// TIA Portal V18 export
FUNCTION_BLOCK "TD_Control"   // FB19, LAD
TITLE = TD_Control
{ S7_Optimized_Access := 'TRUE' }
// Written BY Kristopher Gimenez Feb1,2023
// This block is used to control the TD control mode, pump outputs and HSLT/LSHT shifting
// stored: AutoNumber false, MemoryReserve 100, SetENOAutomatically false
   VAR
      AllowShift : Bool;   // Allow speed change
      TD_Mode : Int;   // TD Mode, 0=Drill, 1=DrillRev, 2=MU-S, 3=MU-T, 4= BO, 5 OSC, 6 Bypass
      HSLTShift_TP { S7_SetPoint := 'True'} : TP_TIME;
      LSHTShift_TP { S7_SetPoint := 'True'} : TP_TIME;
      MUSpinComplete : Bool;   // Set once MU spin torq above setpoint
      TDP1FwdSetmA : Real;
      TDP2FwdSetmA : Real;
      TDP1RevSetmA : Real;
      TDP2RevSetmA : Real;
      TorqSetmA : Real;
      TDP1FwdEn : Bool;
      TDP2FwdEn : Bool;
      TDP1RevEn : Bool;
      TDP2RevEn : Bool;
      TorqEn : Bool;
      BypassDelay_TON { S7_SetPoint := 'True'} : TON_TIME;
      BypassRunning_TOF { S7_SetPoint := 'True'} : TOF_TIME;
      HSLT_Sol_Last { S7_SetPoint := 'True'} : Bool;
      LSHT_Sol_Last : Bool;
      AllowRev : Bool;   // Latch that will allow Drill rev if rotary has stopped
      SpeedLimiting : Bool;
      SpeedLimitmAOut : Real;
      SpeedLimitingTrig : Bool;   // Positive Trigger Last cycle value
      MUTorqStart : Bool;
      BOStart : Bool;
      OscStart : Bool;
      MUTorqStart_Trig : Bool;
      BOStart_Trig : Bool;
      OscStart_Trig : Bool;
      SpeedLimit_SlewDec { S7_SetPoint := 'True'} : "SlewDec";
      SpeedLimit_SlewInc { S7_SetPoint := 'True'} : "SlewInc";
      HiTempShutDown_TON { S7_SetPoint := 'True'} : TON_TIME;
   END_VAR
   VAR_TEMP
      FlowmAOutTemp : Real;
      TorqmAOutTemp : Real;
      TorqPSITemp : Real;
      TorquePSI : Real;
      tempReal : Real;
   END_VAR
   VAR CONSTANT
      Disabled : Int := 0;   // TD Mode State Machine
      Drill : Int := 1;   // TD Mode State Machine
      DrillReverse : Int := 2;   // TD Mode State Machine
      MUSpin : Int := 3;   // TD Mode State Machine
      MUTorq : Int := 4;   // TD Mode State Machine
      BO : Int := 5;   // TD Mode State Machine
      Oscillate : Int := 6;   // TD Mode State Machine
      Bypass : Int := 7;   // TD Mode State Machine
   END_VAR
   VAR_TEMP   // added for the SCL form of the ladder/FBD networks
      _w1 : Bool;
      _w2 : Bool;
      _w3 : Bool;
      _w4 : Bool;
   END_VAR
BEGIN

REGION Network 1: Control Mode
   // Determine Control Mode based on Console Inputs and interlocks.
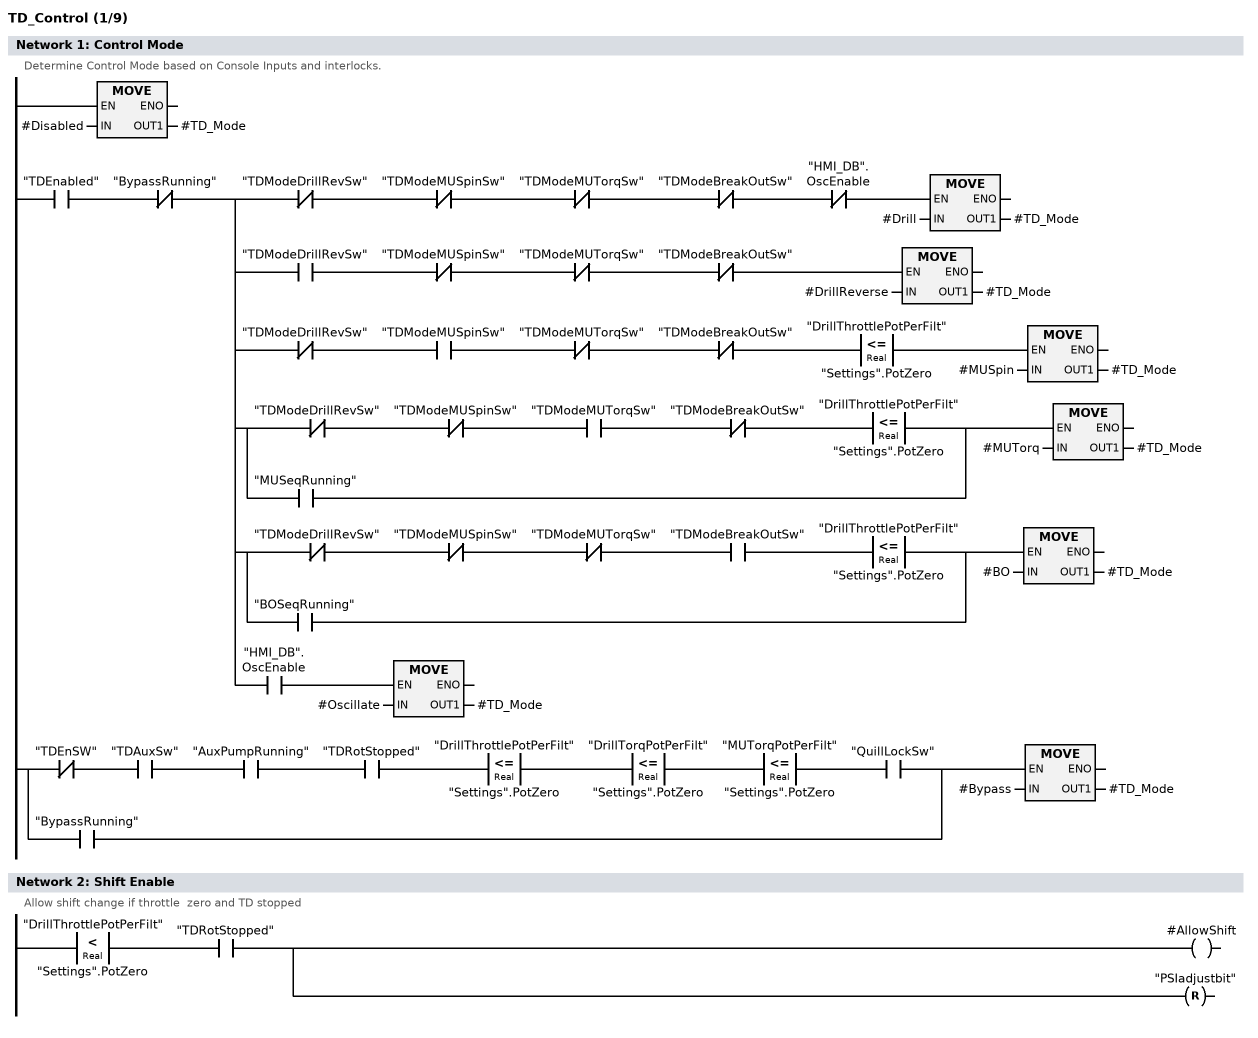
   RUNG wire#powerrail
      Move(in := #Disabled, out1 => #TD_Mode)
   END_RUNG
   RUNG wire#powerrail
      Contact( "TDEnabled" )
      I_Contact( "BypassRunning" )
      wire#w1
      I_Contact( "TDModeDrillRevSw" )
      I_Contact( "TDModeMUSpinSw" )
      I_Contact( "TDModeMUTorqSw" )
      I_Contact( "TDModeBreakOutSw" )
      I_Contact( "HMI_DB".OscEnable )
      Move(in := #Drill, out1 => #TD_Mode)
   END_RUNG
   RUNG wire#w1
      Contact( "TDModeDrillRevSw" )
      I_Contact( "TDModeMUSpinSw" )
      I_Contact( "TDModeMUTorqSw" )
      I_Contact( "TDModeBreakOutSw" )
      Move(in := #DrillReverse, out1 => #TD_Mode)
   END_RUNG
   RUNG wire#w1
      I_Contact( "TDModeDrillRevSw" )
      Contact( "TDModeMUSpinSw" )
      I_Contact( "TDModeMUTorqSw" )
      I_Contact( "TDModeBreakOutSw" )
      { S7_Templates := "SrcType := Real" } LE_Contact(in1 := "DrillThrottlePotPerFilt", in2 := "Settings".PotZero)
      Move(in := #MUSpin, out1 => #TD_Mode)
   END_RUNG
   RUNG wire#w1
      I_Contact( "TDModeDrillRevSw" )
      I_Contact( "TDModeMUSpinSw" )
      Contact( "TDModeMUTorqSw" )
      I_Contact( "TDModeBreakOutSw" )
      { S7_Templates := "SrcType := Real" } LE_Contact(in1 := "DrillThrottlePotPerFilt", in2 := "Settings".PotZero)
      wire#w2
      Move(in := #MUTorq, out1 => #TD_Mode)
   END_RUNG
   RUNG wire#w1
      Contact( "MUSeqRunning" )
   END_RUNG wire#w2
   RUNG wire#w1
      I_Contact( "TDModeDrillRevSw" )
      I_Contact( "TDModeMUSpinSw" )
      I_Contact( "TDModeMUTorqSw" )
      Contact( "TDModeBreakOutSw" )
      { S7_Templates := "SrcType := Real" } LE_Contact(in1 := "DrillThrottlePotPerFilt", in2 := "Settings".PotZero)
      wire#w3
      Move(in := #BO, out1 => #TD_Mode)
   END_RUNG
   RUNG wire#w1
      Contact( "BOSeqRunning" )
   END_RUNG wire#w3
   RUNG wire#w1
      Contact( "HMI_DB".OscEnable )
      Move(in := #Oscillate, out1 => #TD_Mode)
   END_RUNG
   RUNG wire#powerrail
      I_Contact( "TDEnSW" )
      Contact( "TDAuxSw" )
      Contact( "AuxPumpRunning" )
      Contact( "TDRotStopped" )
      { S7_Templates := "SrcType := Real" } LE_Contact(in1 := "DrillThrottlePotPerFilt", in2 := "Settings".PotZero)
      { S7_Templates := "SrcType := Real" } LE_Contact(in1 := "DrillTorqPotPerFilt", in2 := "Settings".PotZero)
      { S7_Templates := "SrcType := Real" } LE_Contact(in1 := "MUTorqPotPerFilt", in2 := "Settings".PotZero)
      Contact( "QuillLockSw" )
      wire#w4
      Move(in := #Bypass, out1 => #TD_Mode)
   END_RUNG
   RUNG wire#powerrail
      Contact( "BypassRunning" )
   END_RUNG wire#w4
   // the same network as SCL:
   #TD_Mode := #Disabled;
   #_w1 := "TDEnabled" AND NOT "BypassRunning";
   IF #_w1 AND NOT "TDModeDrillRevSw" AND NOT "TDModeMUSpinSw" AND NOT "TDModeMUTorqSw" AND NOT "TDModeBreakOutSw" AND NOT "HMI_DB".OscEnable THEN
       #TD_Mode := #Drill;
   END_IF;
   IF #_w1 AND "TDModeDrillRevSw" AND NOT "TDModeMUSpinSw" AND NOT "TDModeMUTorqSw" AND NOT "TDModeBreakOutSw" THEN
       #TD_Mode := #DrillReverse;
   END_IF;
   IF #_w1 AND NOT "TDModeDrillRevSw" AND "TDModeMUSpinSw" AND NOT "TDModeMUTorqSw" AND NOT "TDModeBreakOutSw" AND ("DrillThrottlePotPerFilt" <= "Settings".PotZero) THEN
       #TD_Mode := #MUSpin;
   END_IF;
   IF #_w1 AND ((NOT "TDModeDrillRevSw" AND NOT "TDModeMUSpinSw" AND "TDModeMUTorqSw" AND NOT "TDModeBreakOutSw" AND ("DrillThrottlePotPerFilt" <= "Settings".PotZero)) OR "MUSeqRunning") THEN
       #TD_Mode := #MUTorq;
   END_IF;
   IF #_w1 AND ((NOT "TDModeDrillRevSw" AND NOT "TDModeMUSpinSw" AND NOT "TDModeMUTorqSw" AND "TDModeBreakOutSw" AND ("DrillThrottlePotPerFilt" <= "Settings".PotZero)) OR "BOSeqRunning") THEN
       #TD_Mode := #BO;
   END_IF;
   IF #_w1 AND "HMI_DB".OscEnable THEN #TD_Mode := #Oscillate; END_IF;
   IF (NOT "TDEnSW" AND "TDAuxSw" AND "AuxPumpRunning" AND "TDRotStopped" AND ("DrillThrottlePotPerFilt" <= "Settings".PotZero) AND ("DrillTorqPotPerFilt" <= "Settings".PotZero) AND ("MUTorqPotPerFilt" <= "Settings".PotZero) AND "QuillLockSw") OR "BypassRunning" THEN
       #TD_Mode := #Bypass;
   END_IF;
END_REGION

REGION Network 2: Shift Enable
   // Allow shift change if throttle  zero and TD stopped
   RUNG wire#powerrail
      { S7_Templates := "SrcType := Real" } LT_Contact(in1 := "DrillThrottlePotPerFilt", in2 := "Settings".PotZero)
      Contact( "TDRotStopped" )
      wire#w1
      Coil( #AllowShift )
   END_RUNG
   RUNG wire#w1
      R_Coil( "PSIadjustbit" )
   END_RUNG
   // the same network as SCL:
   #AllowShift := ("DrillThrottlePotPerFilt" < "Settings".PotZero) AND "TDRotStopped";
   IF #AllowShift THEN "PSIadjustbit" := FALSE; END_IF;
END_REGION

REGION Network 3: HSLT/LSHT
   // Allow Shifting.  
   // Bypass in HSLT.  
   // MU modes, BO and Osc in LSHT. 
   // Drill modes follow console input
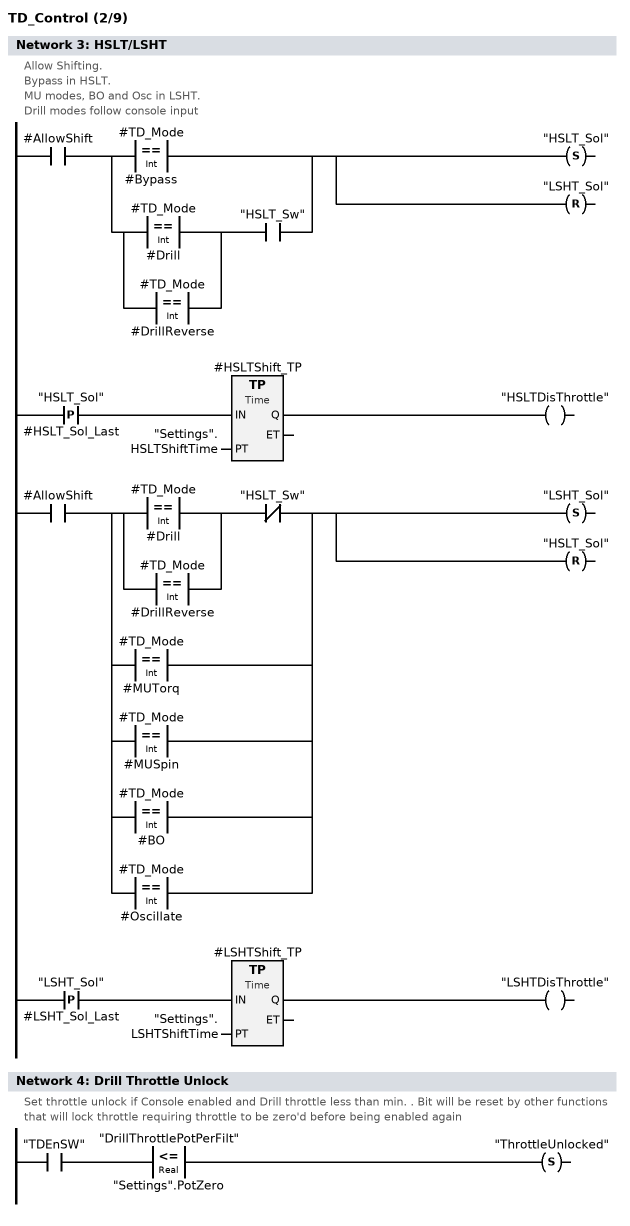
   RUNG wire#powerrail
      Contact( #AllowShift )
      wire#w1
      { S7_Templates := "SrcType := Int" } EQ_Contact(in1 := #TD_Mode, in2 := #Bypass)
      wire#w2
      S_Coil( "HSLT_Sol" )
   END_RUNG
   RUNG wire#w1
      { S7_Templates := "SrcType := Int" } EQ_Contact(in1 := #TD_Mode, in2 := #Drill)
      wire#w3
      Contact( "HSLT_Sw" )
   END_RUNG wire#w2
   RUNG wire#w1
      { S7_Templates := "SrcType := Int" } EQ_Contact(in1 := #TD_Mode, in2 := #DrillReverse)
   END_RUNG wire#w3
   RUNG wire#w2
      R_Coil( "LSHT_Sol" )
   END_RUNG
   RUNG wire#powerrail
      P_Contact(operand := "HSLT_Sol", bit := #HSLT_Sol_Last)
      { S7_Templates := "time_type := Time" } #HSLTShift_TP.TP(pt := "Settings".HSLTShiftTime, et =>)
      Coil( "HSLTDisThrottle" )
   END_RUNG
   RUNG wire#powerrail
      Contact( #AllowShift )
      wire#w4
      { S7_Templates := "SrcType := Int" } EQ_Contact(in1 := #TD_Mode, in2 := #Drill)
      wire#w5
      I_Contact( "HSLT_Sw" )
      wire#w6
      S_Coil( "LSHT_Sol" )
   END_RUNG
   RUNG wire#w4
      { S7_Templates := "SrcType := Int" } EQ_Contact(in1 := #TD_Mode, in2 := #DrillReverse)
   END_RUNG wire#w5
   RUNG wire#w4
      { S7_Templates := "SrcType := Int" } EQ_Contact(in1 := #TD_Mode, in2 := #MUTorq)
   END_RUNG wire#w6
   RUNG wire#w4
      { S7_Templates := "SrcType := Int" } EQ_Contact(in1 := #TD_Mode, in2 := #MUSpin)
   END_RUNG wire#w6
   RUNG wire#w4
      { S7_Templates := "SrcType := Int" } EQ_Contact(in1 := #TD_Mode, in2 := #BO)
   END_RUNG wire#w6
   RUNG wire#w4
      { S7_Templates := "SrcType := Int" } EQ_Contact(in1 := #TD_Mode, in2 := #Oscillate)
   END_RUNG wire#w6
   RUNG wire#w6
      R_Coil( "HSLT_Sol" )
   END_RUNG
   RUNG wire#powerrail
      P_Contact(operand := "LSHT_Sol", bit := #LSHT_Sol_Last)
      { S7_Templates := "time_type := Time" } #LSHTShift_TP.TP(pt := "Settings".LSHTShiftTime, et =>)
      Coil( "LSHTDisThrottle" )
   END_RUNG
   // the same network as SCL:
   IF #AllowShift AND ((#TD_Mode = #Bypass) OR (((#TD_Mode = #Drill) OR (#TD_Mode = #DrillReverse)) AND "HSLT_Sw")) THEN
       "HSLT_Sol" := TRUE;
       "LSHT_Sol" := FALSE;
   END_IF;
   #_w1 := "HSLT_Sol" AND NOT #HSLT_Sol_Last;   // rising edge of "HSLT_Sol"
   #HSLT_Sol_Last := "HSLT_Sol";
   #HSLTShift_TP(IN := #_w1, PT := "Settings".HSLTShiftTime);   // TP
   "HSLTDisThrottle" := #HSLTShift_TP.Q;
   IF #AllowShift AND ((((#TD_Mode = #Drill) OR (#TD_Mode = #DrillReverse)) AND NOT "HSLT_Sw") OR (#TD_Mode = #MUTorq) OR (#TD_Mode = #MUSpin) OR (#TD_Mode = #BO) OR (#TD_Mode = #Oscillate)) THEN
       "LSHT_Sol" := TRUE;
       "HSLT_Sol" := FALSE;
   END_IF;
   #_w2 := "LSHT_Sol" AND NOT #LSHT_Sol_Last;   // rising edge of "LSHT_Sol"
   #LSHT_Sol_Last := "LSHT_Sol";
   #LSHTShift_TP(IN := #_w2, PT := "Settings".LSHTShiftTime);   // TP
   "LSHTDisThrottle" := #LSHTShift_TP.Q;
END_REGION

REGION Network 4: Drill Throttle Unlock
   // Set throttle unlock if Console enabled and Drill throttle less than min. . Bit will be reset by other functions that will lock throttle requiring throttle to be zero'd before being enabled again
   RUNG wire#powerrail
      Contact( "TDEnSW" )
      { S7_Templates := "SrcType := Real" } LE_Contact(in1 := "DrillThrottlePotPerFilt", in2 := "Settings".PotZero)
      S_Coil( "ThrottleUnlocked" )
   END_RUNG
   // the same network as SCL:
   IF "TDEnSW" AND ("DrillThrottlePotPerFilt" <= "Settings".PotZero) THEN "ThrottleUnlocked" := TRUE; END_IF;
END_REGION

REGION Network 5: Drill Throttle Disable
   // Disable throttle if Bypass, Throttle disabled due to shift, or Flush fault or if throttle not unlocked
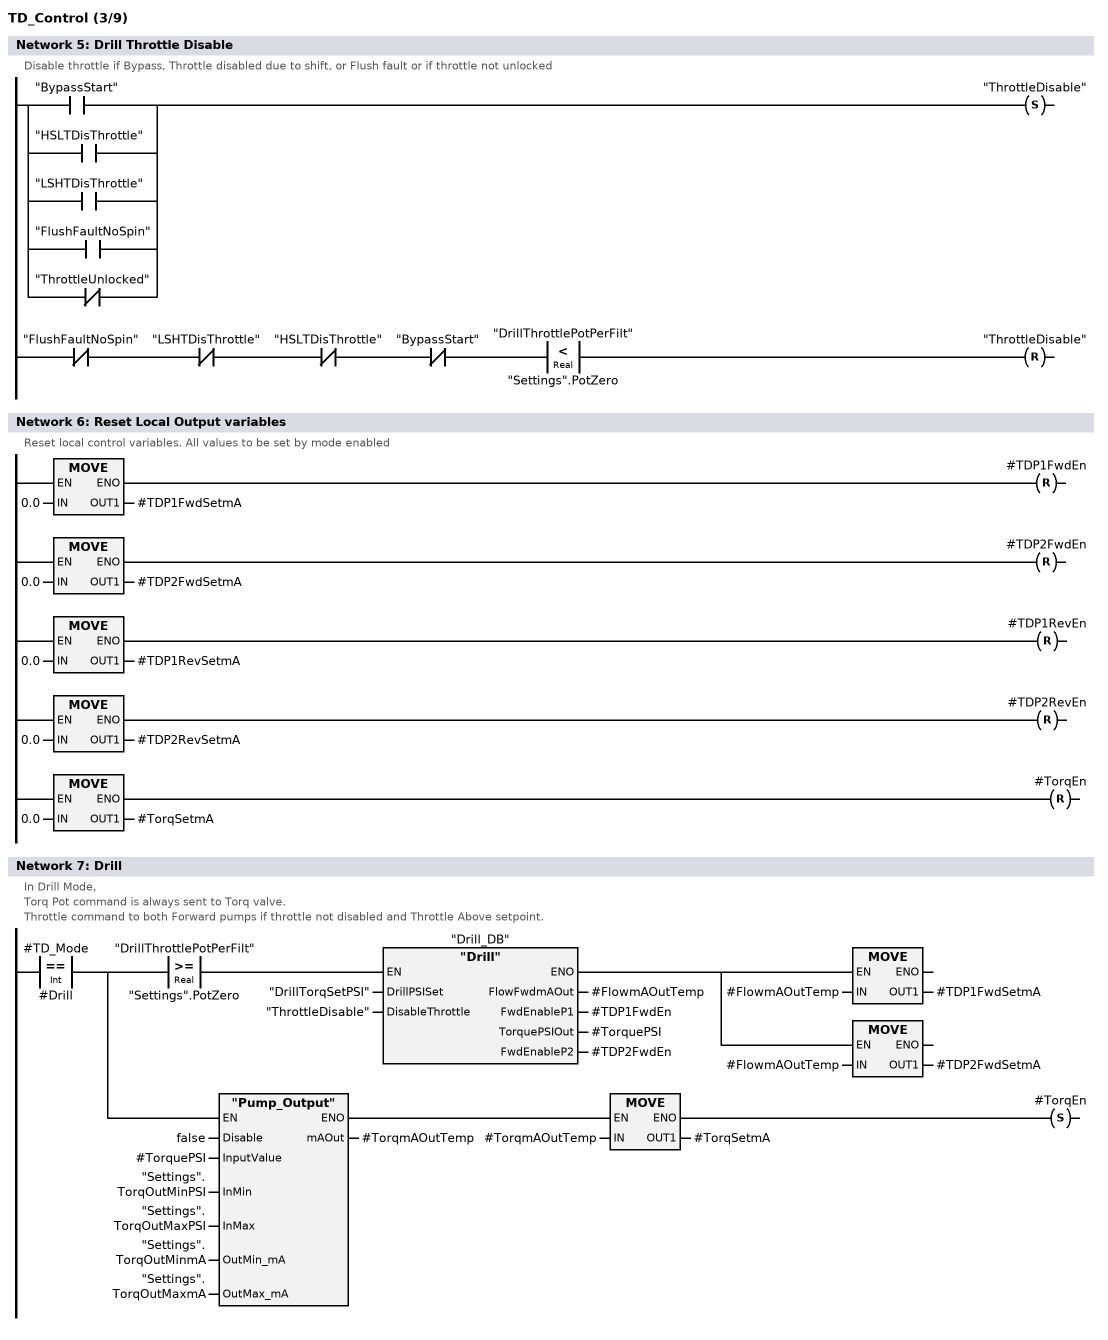
   RUNG wire#powerrail
      Contact( "BypassStart" )
      wire#w1
      S_Coil( "ThrottleDisable" )
   END_RUNG
   RUNG wire#powerrail
      Contact( "HSLTDisThrottle" )
   END_RUNG wire#w1
   RUNG wire#powerrail
      Contact( "LSHTDisThrottle" )
   END_RUNG wire#w1
   RUNG wire#powerrail
      Contact( "FlushFaultNoSpin" )
   END_RUNG wire#w1
   RUNG wire#powerrail
      I_Contact( "ThrottleUnlocked" )
   END_RUNG wire#w1
   RUNG wire#powerrail
      I_Contact( "FlushFaultNoSpin" )
      I_Contact( "LSHTDisThrottle" )
      I_Contact( "HSLTDisThrottle" )
      I_Contact( "BypassStart" )
      { S7_Templates := "SrcType := Real" } LT_Contact(in1 := "DrillThrottlePotPerFilt", in2 := "Settings".PotZero)
      R_Coil( "ThrottleDisable" )
   END_RUNG
   // the same network as SCL:
   IF "BypassStart" OR "HSLTDisThrottle" OR "LSHTDisThrottle" OR "FlushFaultNoSpin" OR NOT "ThrottleUnlocked" THEN
       "ThrottleDisable" := TRUE;
   END_IF;
   IF NOT "FlushFaultNoSpin" AND NOT "LSHTDisThrottle" AND NOT "HSLTDisThrottle" AND NOT "BypassStart" AND ("DrillThrottlePotPerFilt" < "Settings".PotZero) THEN
       "ThrottleDisable" := FALSE;
   END_IF;
END_REGION

REGION Network 6: Reset Local Output variables
   // Reset local control variables. All values to be set by mode enabled
   RUNG wire#powerrail
      Move(in := 0.0, out1 => #TDP1FwdSetmA)
      R_Coil( #TDP1FwdEn )
   END_RUNG
   RUNG wire#powerrail
      Move(in := 0.0, out1 => #TDP2FwdSetmA)
      R_Coil( #TDP2FwdEn )
   END_RUNG
   RUNG wire#powerrail
      Move(in := 0.0, out1 => #TDP1RevSetmA)
      R_Coil( #TDP1RevEn )
   END_RUNG
   RUNG wire#powerrail
      Move(in := 0.0, out1 => #TDP2RevSetmA)
      R_Coil( #TDP2RevEn )
   END_RUNG
   RUNG wire#powerrail
      Move(in := 0.0, out1 => #TorqSetmA)
      R_Coil( #TorqEn )
   END_RUNG
   // the same network as SCL:
   #TDP1FwdSetmA := 0.0;
   #TDP1FwdEn := FALSE;
   #TDP2FwdSetmA := 0.0;
   #TDP2FwdEn := FALSE;
   #TDP1RevSetmA := 0.0;
   #TDP1RevEn := FALSE;
   #TDP2RevSetmA := 0.0;
   #TDP2RevEn := FALSE;
   #TorqSetmA := 0.0;
   #TorqEn := FALSE;
END_REGION

REGION Network 7: Drill
   // In Drill Mode,
   // Torq Pot command is always sent to Torq valve. 
   // Throttle command to both Forward pumps if throttle not disabled and Throttle Above setpoint.
   RUNG wire#powerrail
      { S7_Templates := "SrcType := Int" } EQ_Contact(in1 := #TD_Mode, in2 := #Drill)
      wire#w1
      { S7_Templates := "SrcType := Real" } GE_Contact(in1 := "DrillThrottlePotPerFilt", in2 := "Settings".PotZero)
      "Drill_DB"(DrillPSISet := "DrillTorqSetPSI", DisableThrottle := "ThrottleDisable", FlowFwdmAOut => #FlowmAOutTemp, FwdEnableP1 => #TDP1FwdEn, TorquePSIOut => #TorquePSI, FwdEnableP2 => #TDP2FwdEn)
      wire#w2
      Move(in := #FlowmAOutTemp, out1 => #TDP1FwdSetmA)
   END_RUNG
   RUNG wire#w2
      Move(in := #FlowmAOutTemp, out1 => #TDP2FwdSetmA)
   END_RUNG
   RUNG wire#w1
      "Pump_Output"(Disable := false, InputValue := #TorquePSI, InMin := "Settings".TorqOutMinPSI, InMax := "Settings".TorqOutMaxPSI, OutMin_mA := "Settings".TorqOutMinmA, OutMax_mA := "Settings".TorqOutMaxmA, mAOut => #TorqmAOutTemp)
      Move(in := #TorqmAOutTemp, out1 => #TorqSetmA)
      S_Coil( #TorqEn )
   END_RUNG
   // the same network as SCL:
   #_w1 := #TD_Mode = #Drill;
   "Drill_DB"(EN := #_w1 AND ("DrillThrottlePotPerFilt" >= "Settings".PotZero),   // "Drill"
              DrillPSISet := "DrillTorqSetPSI",
              DisableThrottle := "ThrottleDisable",
              FlowFwdmAOut => #FlowmAOutTemp,
              FwdEnableP1 => #TDP1FwdEn,
              TorquePSIOut => #TorquePSI,
              FwdEnableP2 => #TDP2FwdEn,
              ENO => #_w2);
   IF #_w2 THEN
       #TDP1FwdSetmA := #FlowmAOutTemp;
       #TDP2FwdSetmA := #FlowmAOutTemp;
   END_IF;
   "Pump_Output"(EN := #_w1,
                 Disable := false,
                 InputValue := #TorquePSI,
                 InMin := "Settings".TorqOutMinPSI,
                 InMax := "Settings".TorqOutMaxPSI,
                 OutMin_mA := "Settings".TorqOutMinmA,
                 OutMax_mA := "Settings".TorqOutMaxmA,
                 mAOut => #TorqmAOutTemp,
                 ENO => #_w3);
   IF #_w3 THEN
       #TorqSetmA := #TorqmAOutTemp;
       #TorqEn := TRUE;
   END_IF;
END_REGION

REGION Network 8: Drill Reverse
   // Only allow reverse if TD has stopped moving forward and Throttle above zero. No torq control in reverse. Set at relief
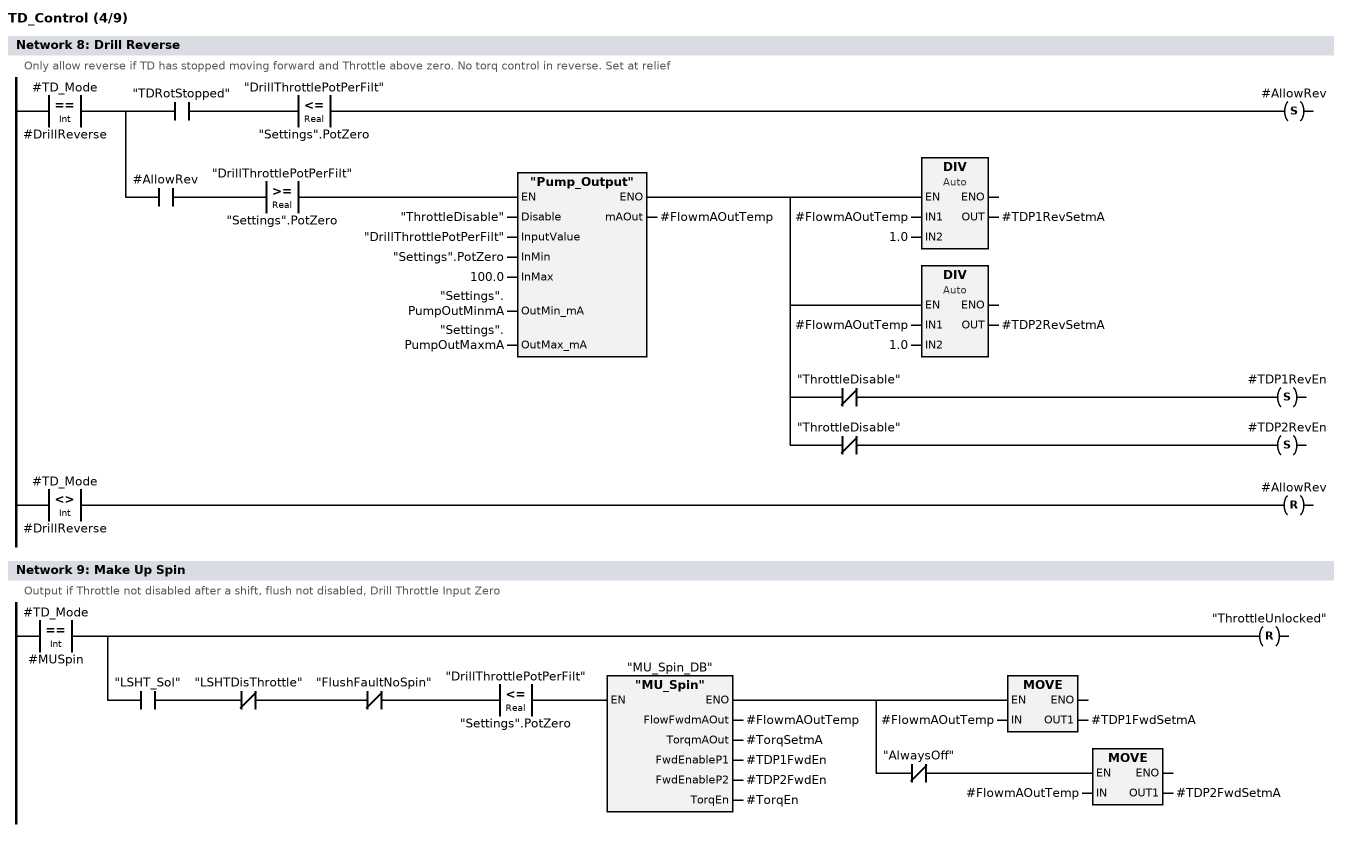
   RUNG wire#powerrail
      { S7_Templates := "SrcType := Int" } EQ_Contact(in1 := #TD_Mode, in2 := #DrillReverse)
      wire#w1
      Contact( "TDRotStopped" )
      { S7_Templates := "SrcType := Real" } LE_Contact(in1 := "DrillThrottlePotPerFilt", in2 := "Settings".PotZero)
      S_Coil( #AllowRev )
   END_RUNG
   RUNG wire#w1
      Contact( #AllowRev )
      { S7_Templates := "SrcType := Real" } GE_Contact(in1 := "DrillThrottlePotPerFilt", in2 := "Settings".PotZero)
      "Pump_Output"(Disable := "ThrottleDisable", InputValue := "DrillThrottlePotPerFilt", InMin := "Settings".PotZero, InMax := 100.0, OutMin_mA := "Settings".PumpOutMinmA, OutMax_mA := "Settings".PumpOutMaxmA, mAOut => #FlowmAOutTemp)
      wire#w2
      Div(in1 := #FlowmAOutTemp, in2 := 1.0, out => #TDP1RevSetmA)
   END_RUNG
   RUNG wire#w2
      Div(in1 := #FlowmAOutTemp, in2 := 1.0, out => #TDP2RevSetmA)
   END_RUNG
   RUNG wire#w2
      I_Contact( "ThrottleDisable" )
      S_Coil( #TDP1RevEn )
   END_RUNG
   RUNG wire#w2
      I_Contact( "ThrottleDisable" )
      S_Coil( #TDP2RevEn )
   END_RUNG
   RUNG wire#powerrail
      { S7_Templates := "SrcType := Int" } NE_Contact(in1 := #TD_Mode, in2 := #DrillReverse)
      R_Coil( #AllowRev )
   END_RUNG
   // the same network as SCL:
   #_w1 := #TD_Mode = #DrillReverse;
   IF #_w1 AND "TDRotStopped" AND ("DrillThrottlePotPerFilt" <= "Settings".PotZero) THEN
       #AllowRev := TRUE;
   END_IF;
   "Pump_Output"(EN := #_w1 AND #AllowRev AND ("DrillThrottlePotPerFilt" >= "Settings".PotZero),
                 Disable := "ThrottleDisable",
                 InputValue := "DrillThrottlePotPerFilt",
                 InMin := "Settings".PotZero,
                 InMax := 100.0,
                 OutMin_mA := "Settings".PumpOutMinmA,
                 OutMax_mA := "Settings".PumpOutMaxmA,
                 mAOut => #FlowmAOutTemp,
                 ENO => #_w2);
   IF #_w2 THEN
       #TDP1RevSetmA := #FlowmAOutTemp / 1.0;
       #TDP2RevSetmA := #FlowmAOutTemp / 1.0;
   END_IF;
   IF #_w2 AND NOT "ThrottleDisable" THEN
       #TDP1RevEn := TRUE;
       #TDP2RevEn := TRUE;
   END_IF;
   IF #TD_Mode <> #DrillReverse THEN #AllowRev := FALSE; END_IF;
END_REGION

REGION Network 9: Make Up Spin
   // Output if Throttle not disabled after a shift, flush not disabled, Drill Throttle Input Zero
   RUNG wire#powerrail
      { S7_Templates := "SrcType := Int" } EQ_Contact(in1 := #TD_Mode, in2 := #MUSpin)
      wire#w1
      R_Coil( "ThrottleUnlocked" )
   END_RUNG
   RUNG wire#w1
      Contact( "LSHT_Sol" )
      I_Contact( "LSHTDisThrottle" )
      I_Contact( "FlushFaultNoSpin" )
      { S7_Templates := "SrcType := Real" } LE_Contact(in1 := "DrillThrottlePotPerFilt", in2 := "Settings".PotZero)
      "MU_Spin_DB"(FlowFwdmAOut => #FlowmAOutTemp, TorqmAOut => #TorqSetmA, FwdEnableP1 => #TDP1FwdEn, FwdEnableP2 => #TDP2FwdEn, TorqEn => #TorqEn)
      wire#w2
      Move(in := #FlowmAOutTemp, out1 => #TDP1FwdSetmA)
   END_RUNG
   RUNG wire#w2
      I_Contact( "AlwaysOff" )
      Move(in := #FlowmAOutTemp, out1 => #TDP2FwdSetmA)
   END_RUNG
   // the same network as SCL:
   #_w1 := #TD_Mode = #MUSpin;
   IF #_w1 THEN "ThrottleUnlocked" := FALSE; END_IF;
   "MU_Spin_DB"(EN := #_w1 AND "LSHT_Sol" AND NOT "LSHTDisThrottle" AND NOT "FlushFaultNoSpin" AND ("DrillThrottlePotPerFilt" <= "Settings".PotZero),   // "MU_Spin"
                FlowFwdmAOut => #FlowmAOutTemp,
                TorqmAOut => #TorqSetmA,
                FwdEnableP1 => #TDP1FwdEn,
                FwdEnableP2 => #TDP2FwdEn,
                TorqEn => #TorqEn,
                ENO => #_w2);
   IF #_w2 THEN #TDP1FwdSetmA := #FlowmAOutTemp; END_IF;
   IF #_w2 AND NOT "AlwaysOff" THEN #TDP2FwdSetmA := #FlowmAOutTemp; END_IF;
END_REGION

REGION Network 10: Make Up Torque
   // Output if Throttle not disabled after a shift, flush not disabled, Drill Throttle Input Zero
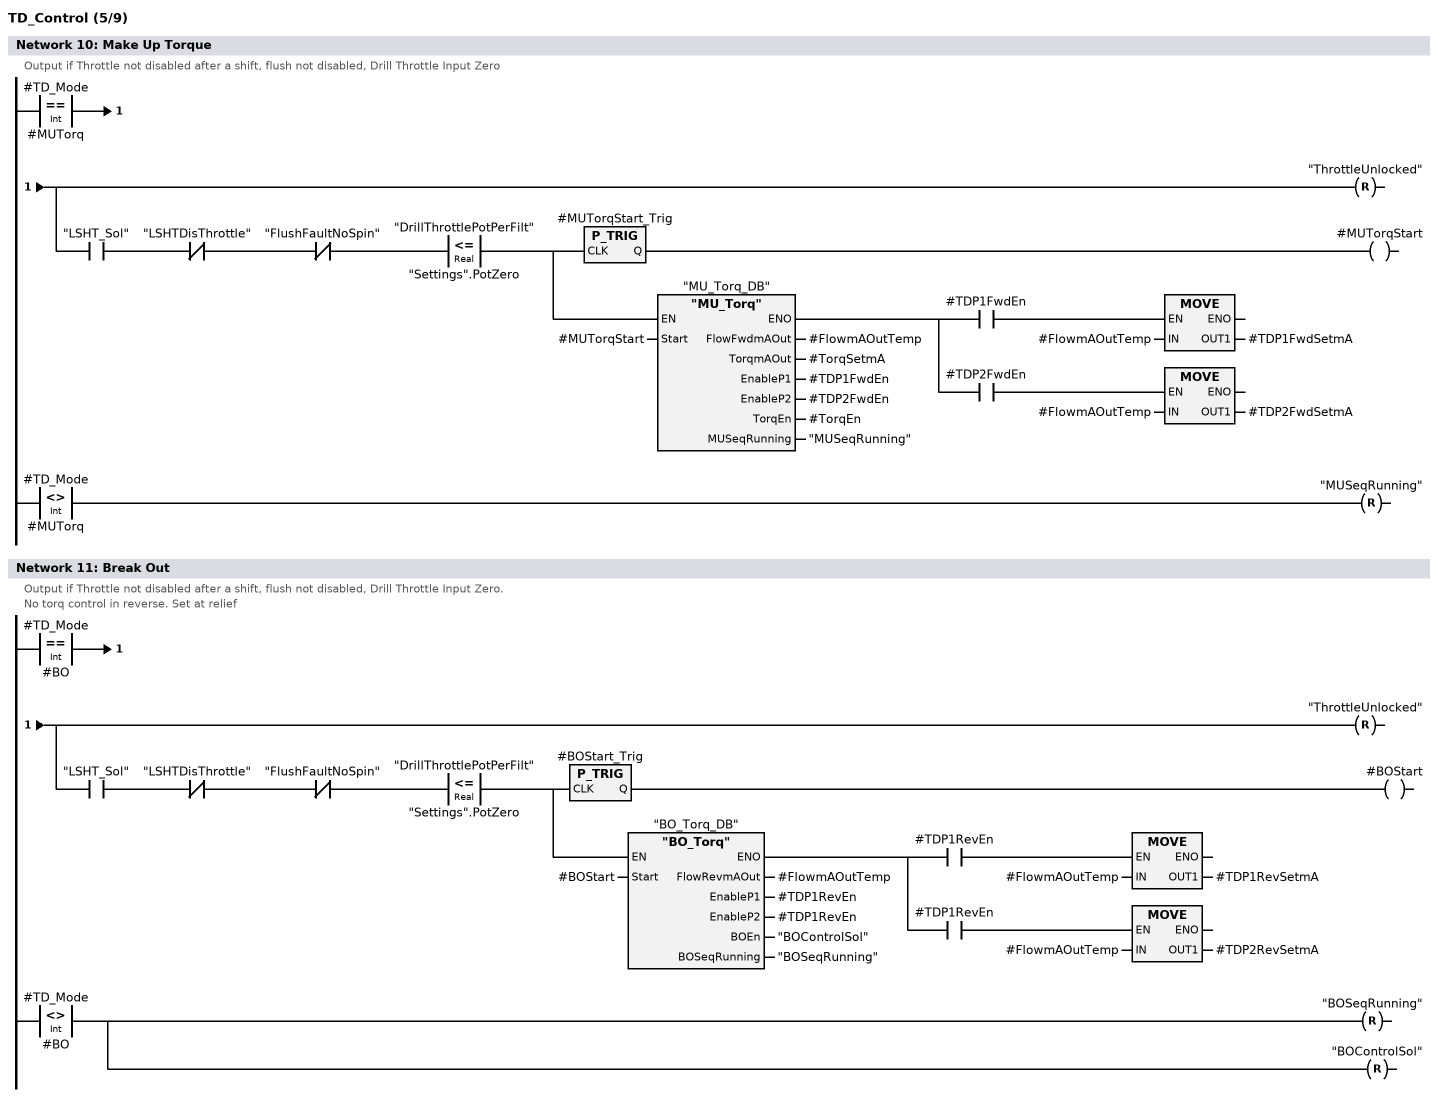
   RUNG wire#powerrail
      { S7_Templates := "SrcType := Int" } EQ_Contact(in1 := #TD_Mode, in2 := #MUTorq)
      wire#w1
      R_Coil( "ThrottleUnlocked" )
   END_RUNG
   RUNG wire#w1
      Contact( "LSHT_Sol" )
      I_Contact( "LSHTDisThrottle" )
      I_Contact( "FlushFaultNoSpin" )
      { S7_Templates := "SrcType := Real" } LE_Contact(in1 := "DrillThrottlePotPerFilt", in2 := "Settings".PotZero)
      wire#w2
      P_Trig( #MUTorqStart_Trig )
      Coil( #MUTorqStart )
   END_RUNG
   RUNG wire#w2
      "MU_Torq_DB"(Start := #MUTorqStart, FlowFwdmAOut => #FlowmAOutTemp, TorqmAOut => #TorqSetmA, EnableP1 => #TDP1FwdEn, EnableP2 => #TDP2FwdEn, TorqEn => #TorqEn, MUSeqRunning => "MUSeqRunning")
      wire#w3
      Contact( #TDP1FwdEn )
      Move(in := #FlowmAOutTemp, out1 => #TDP1FwdSetmA)
   END_RUNG
   RUNG wire#w3
      Contact( #TDP2FwdEn )
      Move(in := #FlowmAOutTemp, out1 => #TDP2FwdSetmA)
   END_RUNG
   RUNG wire#powerrail
      { S7_Templates := "SrcType := Int" } NE_Contact(in1 := #TD_Mode, in2 := #MUTorq)
      R_Coil( "MUSeqRunning" )
   END_RUNG
   // the same network as SCL:
   #_w1 := #TD_Mode = #MUTorq;
   IF #_w1 THEN "ThrottleUnlocked" := FALSE; END_IF;
   #_w2 := #_w1 AND "LSHT_Sol" AND NOT "LSHTDisThrottle" AND NOT "FlushFaultNoSpin" AND ("DrillThrottlePotPerFilt" <= "Settings".PotZero);
   #_w3 := #_w2 AND NOT #MUTorqStart_Trig;   // rising edge
   #MUTorqStart_Trig := #_w2;
   #MUTorqStart := #_w3;
   "MU_Torq_DB"(EN := #_w2,   // "MU_Torq"
                Start := #MUTorqStart,
                FlowFwdmAOut => #FlowmAOutTemp,
                TorqmAOut => #TorqSetmA,
                EnableP1 => #TDP1FwdEn,
                EnableP2 => #TDP2FwdEn,
                TorqEn => #TorqEn,
                MUSeqRunning => "MUSeqRunning",
                ENO => #_w4);
   IF #_w4 AND #TDP1FwdEn THEN #TDP1FwdSetmA := #FlowmAOutTemp; END_IF;
   IF #_w4 AND #TDP2FwdEn THEN #TDP2FwdSetmA := #FlowmAOutTemp; END_IF;
   IF #TD_Mode <> #MUTorq THEN "MUSeqRunning" := FALSE; END_IF;
END_REGION

REGION Network 11: Break Out
   // Output if Throttle not disabled after a shift, flush not disabled, Drill Throttle Input Zero.
   // No torq control in reverse. Set at relief
   RUNG wire#powerrail
      { S7_Templates := "SrcType := Int" } EQ_Contact(in1 := #TD_Mode, in2 := #BO)
      wire#w1
      R_Coil( "ThrottleUnlocked" )
   END_RUNG
   RUNG wire#w1
      Contact( "LSHT_Sol" )
      I_Contact( "LSHTDisThrottle" )
      I_Contact( "FlushFaultNoSpin" )
      { S7_Templates := "SrcType := Real" } LE_Contact(in1 := "DrillThrottlePotPerFilt", in2 := "Settings".PotZero)
      wire#w2
      P_Trig( #BOStart_Trig )
      Coil( #BOStart )
   END_RUNG
   RUNG wire#w2
      "BO_Torq_DB"(Start := #BOStart, FlowRevmAOut => #FlowmAOutTemp, EnableP1 => #TDP1RevEn, EnableP2 => #TDP1RevEn, BOEn => "BOControlSol", BOSeqRunning => "BOSeqRunning")
      wire#w3
      Contact( #TDP1RevEn )
      Move(in := #FlowmAOutTemp, out1 => #TDP1RevSetmA)
   END_RUNG
   RUNG wire#w3
      Contact( #TDP1RevEn )
      Move(in := #FlowmAOutTemp, out1 => #TDP2RevSetmA)
   END_RUNG
   RUNG wire#powerrail
      { S7_Templates := "SrcType := Int" } NE_Contact(in1 := #TD_Mode, in2 := #BO)
      wire#w4
      R_Coil( "BOSeqRunning" )
   END_RUNG
   RUNG wire#w4
      R_Coil( "BOControlSol" )
   END_RUNG
   // the same network as SCL:
   #_w1 := #TD_Mode = #BO;
   IF #_w1 THEN "ThrottleUnlocked" := FALSE; END_IF;
   #_w2 := #_w1 AND "LSHT_Sol" AND NOT "LSHTDisThrottle" AND NOT "FlushFaultNoSpin" AND ("DrillThrottlePotPerFilt" <= "Settings".PotZero);
   #_w3 := #_w2 AND NOT #BOStart_Trig;   // rising edge
   #BOStart_Trig := #_w2;
   #BOStart := #_w3;
   "BO_Torq_DB"(EN := #_w2,   // "BO_Torq"
                Start := #BOStart,
                FlowRevmAOut => #FlowmAOutTemp,
                EnableP1 => #TDP1RevEn,
                EnableP2 => #TDP1RevEn,
                BOEn => "BOControlSol",
                BOSeqRunning => "BOSeqRunning",
                ENO => #_w4);
   IF #_w4 AND #TDP1RevEn THEN
       #TDP1RevSetmA := #FlowmAOutTemp;
       #TDP2RevSetmA := #FlowmAOutTemp;
   END_IF;
   IF #TD_Mode <> #BO THEN
       "BOSeqRunning" := FALSE;
       "BOControlSol" := FALSE;
   END_IF;
END_REGION

REGION Network 12: Oscillator
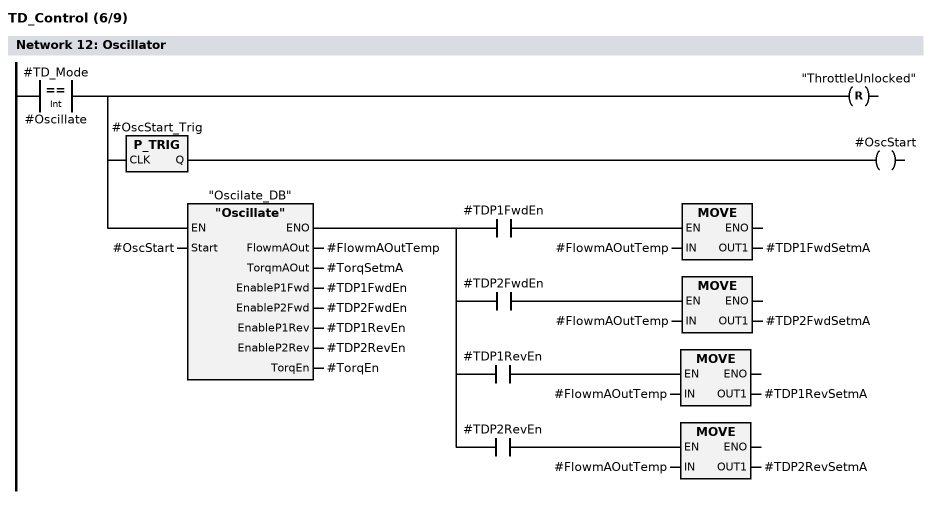
   RUNG wire#powerrail
      { S7_Templates := "SrcType := Int" } EQ_Contact(in1 := #TD_Mode, in2 := #Oscillate)
      wire#w1
      R_Coil( "ThrottleUnlocked" )
   END_RUNG
   RUNG wire#w1
      P_Trig( #OscStart_Trig )
      Coil( #OscStart )
   END_RUNG
   RUNG wire#w1
      "Oscilate_DB"(Start := #OscStart, FlowmAOut => #FlowmAOutTemp, TorqmAOut => #TorqSetmA, EnableP1Fwd => #TDP1FwdEn, EnableP2Fwd => #TDP2FwdEn, EnableP1Rev => #TDP1RevEn, EnableP2Rev => #TDP2RevEn, TorqEn => #TorqEn)
      wire#w2
      Contact( #TDP1FwdEn )
      Move(in := #FlowmAOutTemp, out1 => #TDP1FwdSetmA)
   END_RUNG
   RUNG wire#w2
      Contact( #TDP2FwdEn )
      Move(in := #FlowmAOutTemp, out1 => #TDP2FwdSetmA)
   END_RUNG
   RUNG wire#w2
      Contact( #TDP1RevEn )
      Move(in := #FlowmAOutTemp, out1 => #TDP1RevSetmA)
   END_RUNG
   RUNG wire#w2
      Contact( #TDP2RevEn )
      Move(in := #FlowmAOutTemp, out1 => #TDP2RevSetmA)
   END_RUNG
   // the same network as SCL:
   #_w1 := #TD_Mode = #Oscillate;
   IF #_w1 THEN "ThrottleUnlocked" := FALSE; END_IF;
   #_w2 := #_w1 AND NOT #OscStart_Trig;   // rising edge
   #OscStart_Trig := #_w1;
   #OscStart := #_w2;
   "Oscilate_DB"(EN := #_w1,   // "Oscillate"
                 Start := #OscStart,
                 FlowmAOut => #FlowmAOutTemp,
                 TorqmAOut => #TorqSetmA,
                 EnableP1Fwd => #TDP1FwdEn,
                 EnableP2Fwd => #TDP2FwdEn,
                 EnableP1Rev => #TDP1RevEn,
                 EnableP2Rev => #TDP2RevEn,
                 TorqEn => #TorqEn,
                 ENO => #_w3);
   IF #_w3 AND #TDP1FwdEn THEN #TDP1FwdSetmA := #FlowmAOutTemp; END_IF;
   IF #_w3 AND #TDP2FwdEn THEN #TDP2FwdSetmA := #FlowmAOutTemp; END_IF;
   IF #_w3 AND #TDP1RevEn THEN #TDP1RevSetmA := #FlowmAOutTemp; END_IF;
   IF #_w3 AND #TDP2RevEn THEN #TDP2RevSetmA := #FlowmAOutTemp; END_IF;
END_REGION

REGION Network 13: Bypass Mode
   // In Bypass Mode
   // If gripper closed turn on Bypass valve(Quill is Locked after PTO funtioned)
   // After PTO wait 8 seconds for system to enage before enabling bypass control outputs
   // Note TD in HSLT in Bypass mode
   // Bypass Running flag will stay on for Set time after Bypass mode finished
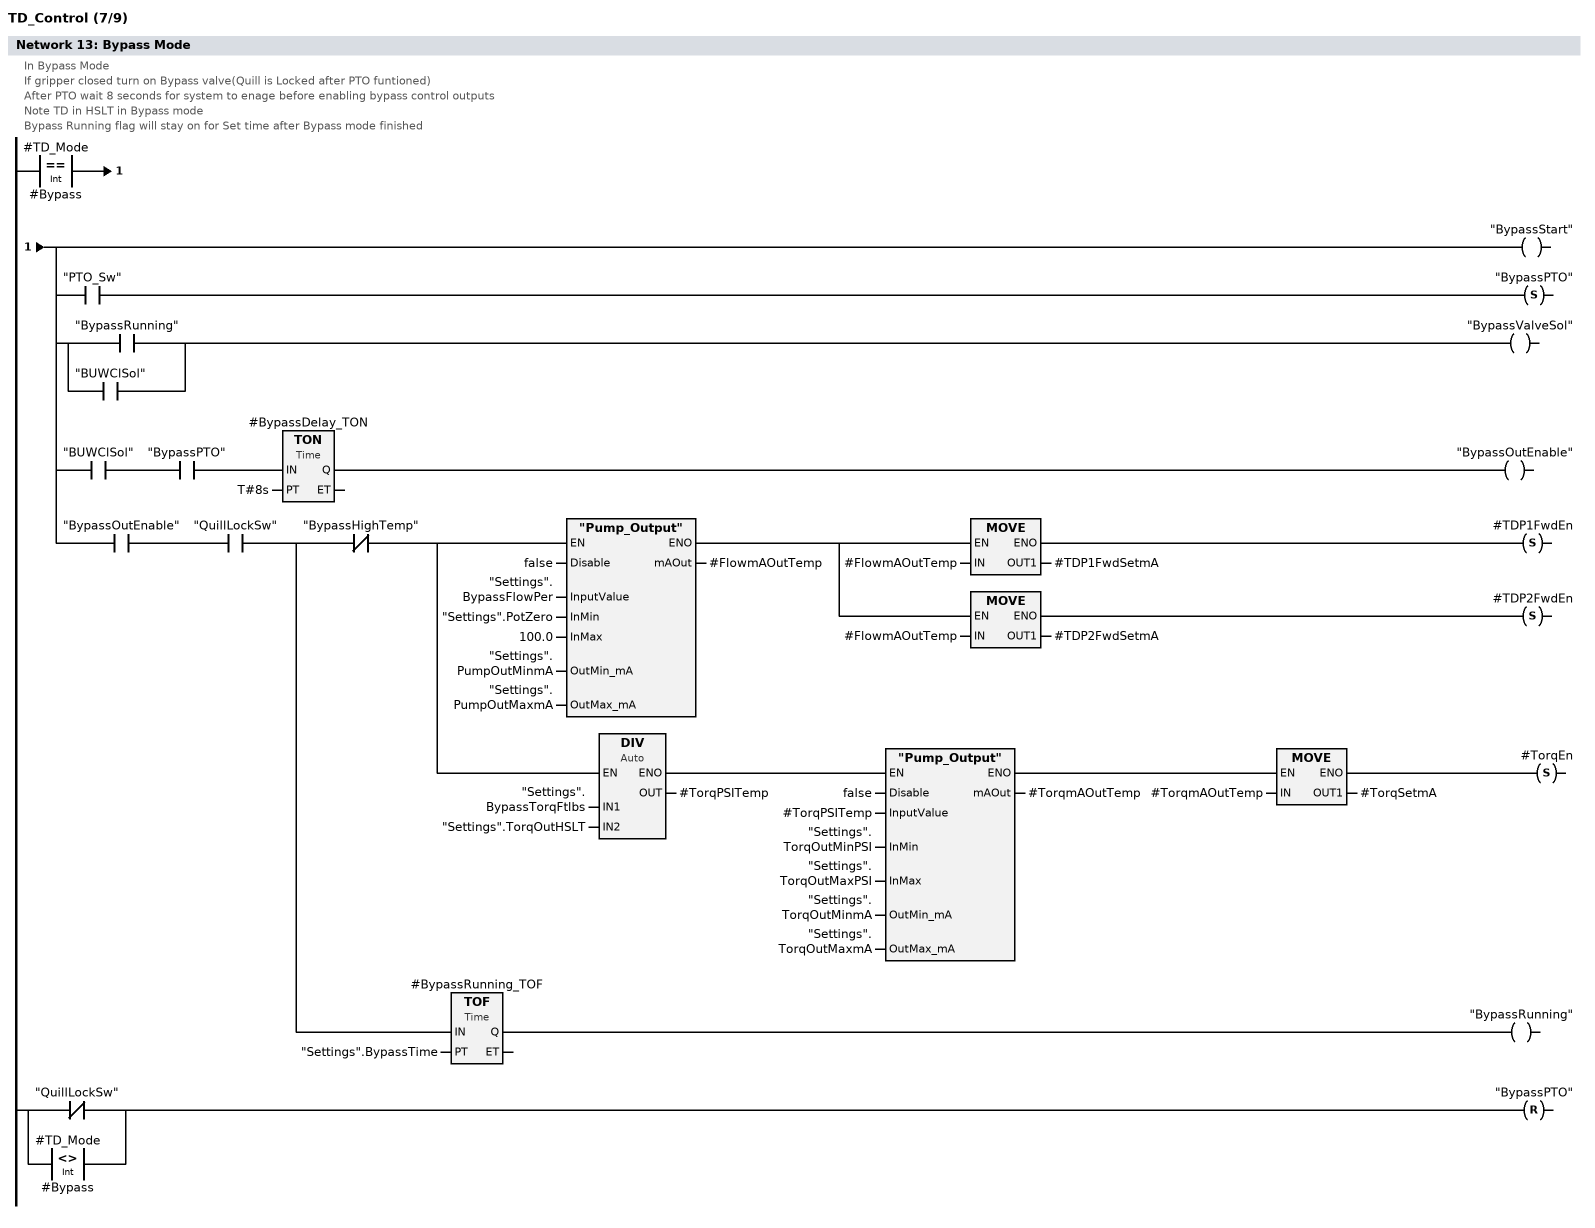
   RUNG wire#powerrail
      { S7_Templates := "SrcType := Int" } EQ_Contact(in1 := #TD_Mode, in2 := #Bypass)
      wire#w1
      Coil( "BypassStart" )
   END_RUNG
   RUNG wire#w1
      Contact( "PTO_Sw" )
      S_Coil( "BypassPTO" )
   END_RUNG
   RUNG wire#w1
      Contact( "BypassRunning" )
      wire#w2
      Coil( "BypassValveSol" )
   END_RUNG
   RUNG wire#w1
      Contact( "BUWClSol" )
   END_RUNG wire#w2
   RUNG wire#w1
      Contact( "BUWClSol" )
      Contact( "BypassPTO" )
      { S7_Templates := "time_type := Time" } #BypassDelay_TON.TON(pt := T#8s, et =>)
      Coil( "BypassOutEnable" )
   END_RUNG
   RUNG wire#w1
      Contact( "BypassOutEnable" )
      Contact( "QuillLockSw" )
      wire#w3
      I_Contact( "BypassHighTemp" )
      wire#w4
      "Pump_Output"(Disable := false, InputValue := "Settings".BypassFlowPer, InMin := "Settings".PotZero, InMax := 100.0, OutMin_mA := "Settings".PumpOutMinmA, OutMax_mA := "Settings".PumpOutMaxmA, mAOut => #FlowmAOutTemp)
      wire#w5
      Move(in := #FlowmAOutTemp, out1 => #TDP1FwdSetmA)
      S_Coil( #TDP1FwdEn )
   END_RUNG
   RUNG wire#w5
      Move(in := #FlowmAOutTemp, out1 => #TDP2FwdSetmA)
      S_Coil( #TDP2FwdEn )
   END_RUNG
   RUNG wire#w4
      Div(in1 := "Settings".BypassTorqFtlbs, in2 := "Settings".TorqOutHSLT, out => #TorqPSITemp)
      "Pump_Output"(Disable := false, InputValue := #TorqPSITemp, InMin := "Settings".TorqOutMinPSI, InMax := "Settings".TorqOutMaxPSI, OutMin_mA := "Settings".TorqOutMinmA, OutMax_mA := "Settings".TorqOutMaxmA, mAOut => #TorqmAOutTemp)
      Move(in := #TorqmAOutTemp, out1 => #TorqSetmA)
      S_Coil( #TorqEn )
   END_RUNG
   RUNG wire#w3
      { S7_Templates := "time_type := Time" } #BypassRunning_TOF.TOF(pt := "Settings".BypassTime, et =>)
      Coil( "BypassRunning" )
   END_RUNG
   RUNG wire#powerrail
      I_Contact( "QuillLockSw" )
      wire#w6
      R_Coil( "BypassPTO" )
   END_RUNG
   RUNG wire#powerrail
      { S7_Templates := "SrcType := Int" } NE_Contact(in1 := #TD_Mode, in2 := #Bypass)
   END_RUNG wire#w6
   // the same network as SCL:
   "BypassStart" := #TD_Mode = #Bypass;
   IF "BypassStart" AND "PTO_Sw" THEN "BypassPTO" := TRUE; END_IF;
   "BypassValveSol" := "BypassStart" AND ("BypassRunning" OR "BUWClSol");
   #BypassDelay_TON(IN := "BypassStart" AND "BUWClSol" AND "BypassPTO", PT := T#8s);   // TON
   "BypassOutEnable" := #BypassDelay_TON.Q;
   #_w1 := "BypassStart" AND "BypassOutEnable" AND "QuillLockSw";
   #_w3 := #_w1 AND NOT "BypassHighTemp";
   "Pump_Output"(EN := #_w1 AND NOT "BypassHighTemp",
                 Disable := false,
                 InputValue := "Settings".BypassFlowPer,
                 InMin := "Settings".PotZero,
                 InMax := 100.0,
                 OutMin_mA := "Settings".PumpOutMinmA,
                 OutMax_mA := "Settings".PumpOutMaxmA,
                 mAOut => #FlowmAOutTemp,
                 ENO => #_w2);
   IF #_w2 THEN
       #TDP1FwdSetmA := #FlowmAOutTemp;
       #TDP1FwdEn := TRUE;
       #TDP2FwdSetmA := #FlowmAOutTemp;
       #TDP2FwdEn := TRUE;
   END_IF;
   IF #_w3 THEN #TorqPSITemp := "Settings".BypassTorqFtlbs / "Settings".TorqOutHSLT; END_IF;
   "Pump_Output"(EN := #_w3,
                 Disable := false,
                 InputValue := #TorqPSITemp,
                 InMin := "Settings".TorqOutMinPSI,
                 InMax := "Settings".TorqOutMaxPSI,
                 OutMin_mA := "Settings".TorqOutMinmA,
                 OutMax_mA := "Settings".TorqOutMaxmA,
                 mAOut => #TorqmAOutTemp,
                 ENO => #_w4);
   IF #_w4 THEN
       #TorqSetmA := #TorqmAOutTemp;
       #TorqEn := TRUE;
   END_IF;
   #BypassRunning_TOF(IN := #_w1, PT := "Settings".BypassTime);   // TOF
   "BypassRunning" := #BypassRunning_TOF.Q;
   IF NOT "QuillLockSw" OR (#TD_Mode <> #Bypass) THEN "BypassPTO" := FALSE; END_IF;
END_REGION

REGION Network 14: Max Speed Limiter
   // Limit Output to Pump if speed above Max Speed Low Setpoint
   // While Limiting, Destroke Output to pump if above Max Speed High Setpoint and increase if below
   // Note In HSLT, drill mode active and both pumps used
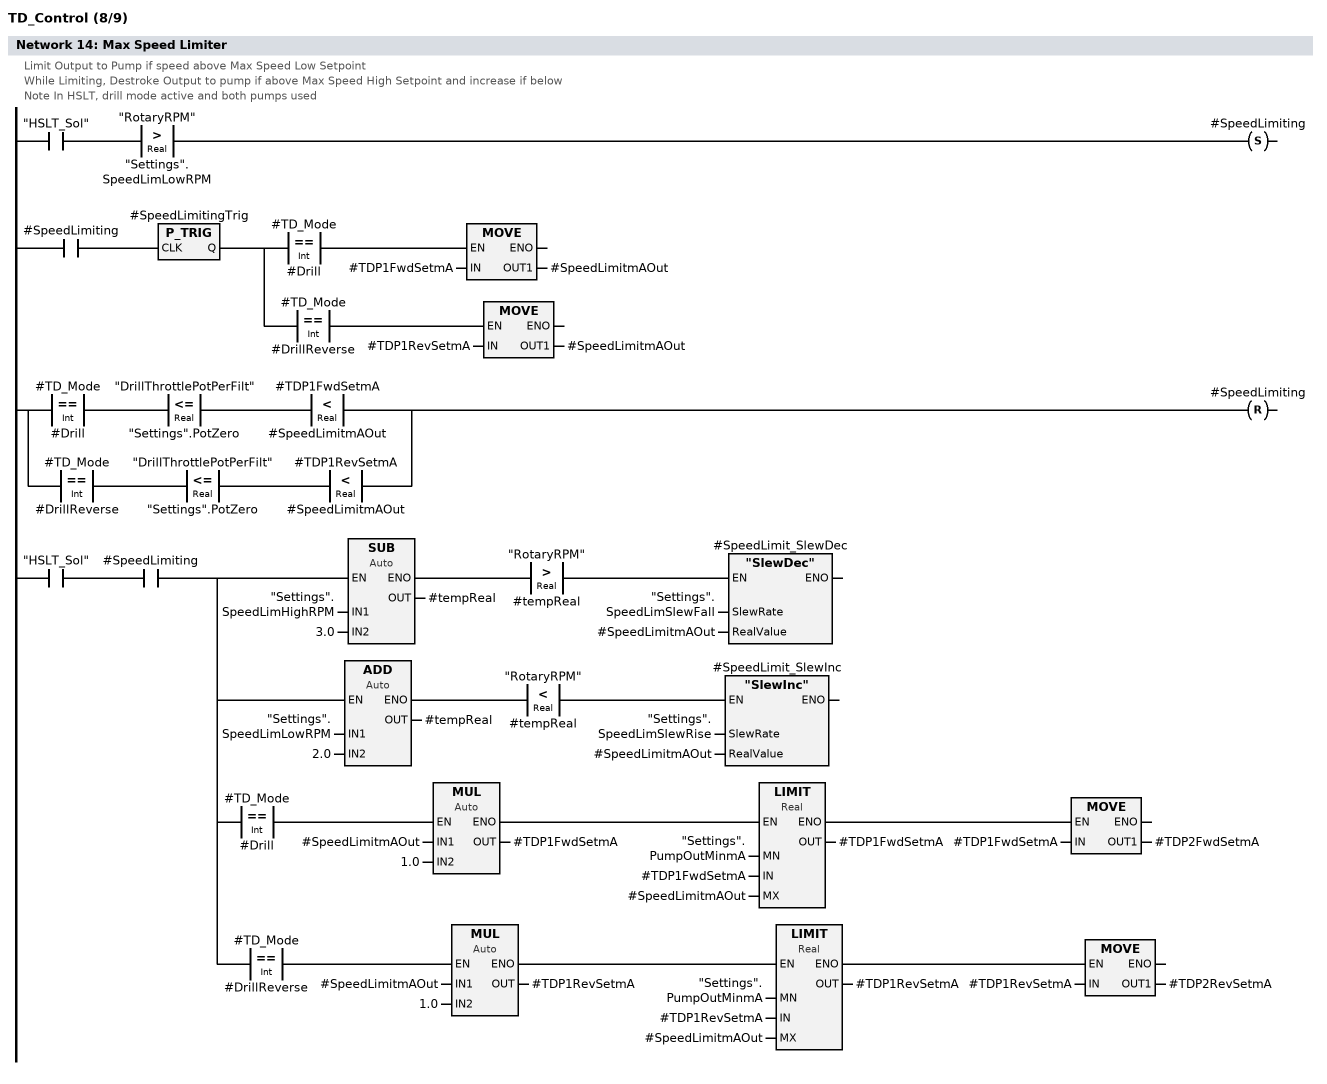
   RUNG wire#powerrail
      Contact( "HSLT_Sol" )
      { S7_Templates := "SrcType := Real" } GT_Contact(in1 := "RotaryRPM", in2 := "Settings".SpeedLimLowRPM)
      S_Coil( #SpeedLimiting )
   END_RUNG
   RUNG wire#powerrail
      Contact( #SpeedLimiting )
      P_Trig( #SpeedLimitingTrig )
      wire#w1
      { S7_Templates := "SrcType := Int" } EQ_Contact(in1 := #TD_Mode, in2 := #Drill)
      Move(in := #TDP1FwdSetmA, out1 => #SpeedLimitmAOut)
   END_RUNG
   RUNG wire#w1
      { S7_Templates := "SrcType := Int" } EQ_Contact(in1 := #TD_Mode, in2 := #DrillReverse)
      Move(in := #TDP1RevSetmA, out1 => #SpeedLimitmAOut)
   END_RUNG
   RUNG wire#powerrail
      { S7_Templates := "SrcType := Int" } EQ_Contact(in1 := #TD_Mode, in2 := #Drill)
      { S7_Templates := "SrcType := Real" } LE_Contact(in1 := "DrillThrottlePotPerFilt", in2 := "Settings".PotZero)
      { S7_Templates := "SrcType := Real" } LT_Contact(in1 := #TDP1FwdSetmA, in2 := #SpeedLimitmAOut)
      wire#w2
      R_Coil( #SpeedLimiting )
   END_RUNG
   RUNG wire#powerrail
      { S7_Templates := "SrcType := Int" } EQ_Contact(in1 := #TD_Mode, in2 := #DrillReverse)
      { S7_Templates := "SrcType := Real" } LE_Contact(in1 := "DrillThrottlePotPerFilt", in2 := "Settings".PotZero)
      { S7_Templates := "SrcType := Real" } LT_Contact(in1 := #TDP1RevSetmA, in2 := #SpeedLimitmAOut)
   END_RUNG wire#w2
   RUNG wire#powerrail
      Contact( "HSLT_Sol" )
      Contact( #SpeedLimiting )
      wire#w3
      Sub(in1 := "Settings".SpeedLimHighRPM, in2 := 3.0, out => #tempReal)
      { S7_Templates := "SrcType := Real" } GT_Contact(in1 := "RotaryRPM", in2 := #tempReal)
      #SpeedLimit_SlewDec(SlewRate := "Settings".SpeedLimSlewFall, RealValue := #SpeedLimitmAOut)
   END_RUNG
   RUNG wire#w3
      Add(in1 := "Settings".SpeedLimLowRPM, in2 := 2.0, out => #tempReal)
      { S7_Templates := "SrcType := Real" } LT_Contact(in1 := "RotaryRPM", in2 := #tempReal)
      #SpeedLimit_SlewInc(SlewRate := "Settings".SpeedLimSlewRise, RealValue := #SpeedLimitmAOut)
   END_RUNG
   RUNG wire#w3
      { S7_Templates := "SrcType := Int" } EQ_Contact(in1 := #TD_Mode, in2 := #Drill)
      Mul(in1 := #SpeedLimitmAOut, in2 := 1.0, out => #TDP1FwdSetmA)
      { S7_Templates := "value_type := Real" } Limit(mn := "Settings".PumpOutMinmA, in := #TDP1FwdSetmA, mx := #SpeedLimitmAOut, out => #TDP1FwdSetmA)
      Move(in := #TDP1FwdSetmA, out1 => #TDP2FwdSetmA)
   END_RUNG
   RUNG wire#w3
      { S7_Templates := "SrcType := Int" } EQ_Contact(in1 := #TD_Mode, in2 := #DrillReverse)
      Mul(in1 := #SpeedLimitmAOut, in2 := 1.0, out => #TDP1RevSetmA)
      { S7_Templates := "value_type := Real" } Limit(mn := "Settings".PumpOutMinmA, in := #TDP1RevSetmA, mx := #SpeedLimitmAOut, out => #TDP1RevSetmA)
      Move(in := #TDP1RevSetmA, out1 => #TDP2RevSetmA)
   END_RUNG
   // the same network as SCL:
   IF "HSLT_Sol" AND ("RotaryRPM" > "Settings".SpeedLimLowRPM) THEN #SpeedLimiting := TRUE; END_IF;
   #_w1 := #SpeedLimiting AND NOT #SpeedLimitingTrig;   // rising edge
   #SpeedLimitingTrig := #SpeedLimiting;
   IF #_w1 AND (#TD_Mode = #Drill) THEN #SpeedLimitmAOut := #TDP1FwdSetmA; END_IF;
   IF #_w1 AND (#TD_Mode = #DrillReverse) THEN #SpeedLimitmAOut := #TDP1RevSetmA; END_IF;
   IF ((#TD_Mode = #Drill) AND ("DrillThrottlePotPerFilt" <= "Settings".PotZero) AND (#TDP1FwdSetmA < #SpeedLimitmAOut)) OR ((#TD_Mode = #DrillReverse) AND ("DrillThrottlePotPerFilt" <= "Settings".PotZero) AND (#TDP1RevSetmA < #SpeedLimitmAOut)) THEN
       #SpeedLimiting := FALSE;
   END_IF;
   #_w2 := "HSLT_Sol" AND #SpeedLimiting;
   IF #_w2 THEN #tempReal := "Settings".SpeedLimHighRPM - 3.0; END_IF;
   IF #_w2 AND ("RotaryRPM" > #tempReal) THEN
       #SpeedLimit_SlewDec(SlewRate := "Settings".SpeedLimSlewFall, RealValue := #SpeedLimitmAOut);   // "SlewDec"
   END_IF;
   IF #_w2 THEN #tempReal := "Settings".SpeedLimLowRPM + 2.0; END_IF;
   IF #_w2 AND ("RotaryRPM" < #tempReal) THEN
       #SpeedLimit_SlewInc(SlewRate := "Settings".SpeedLimSlewRise, RealValue := #SpeedLimitmAOut);   // "SlewInc"
   END_IF;
   IF #_w2 AND (#TD_Mode = #Drill) THEN
       #TDP1FwdSetmA := #SpeedLimitmAOut * 1.0;
       #TDP1FwdSetmA := LIMIT(MN := "Settings".PumpOutMinmA, IN := #TDP1FwdSetmA, MX := #SpeedLimitmAOut);
       #TDP2FwdSetmA := #TDP1FwdSetmA;
   END_IF;
   IF #_w2 AND (#TD_Mode = #DrillReverse) THEN
       #TDP1RevSetmA := #SpeedLimitmAOut * 1.0;
       #TDP1RevSetmA := LIMIT(MN := "Settings".PumpOutMinmA, IN := #TDP1RevSetmA, MX := #SpeedLimitmAOut);
       #TDP2RevSetmA := #TDP1RevSetmA;
   END_IF;
END_REGION

REGION Network 15: High Temp Speed Limiter
   // Limit Flow mA Output if High Temp reduced RPM.
   // 
   // Disable outputs 10 seconds after a shutdown and disable Throttle
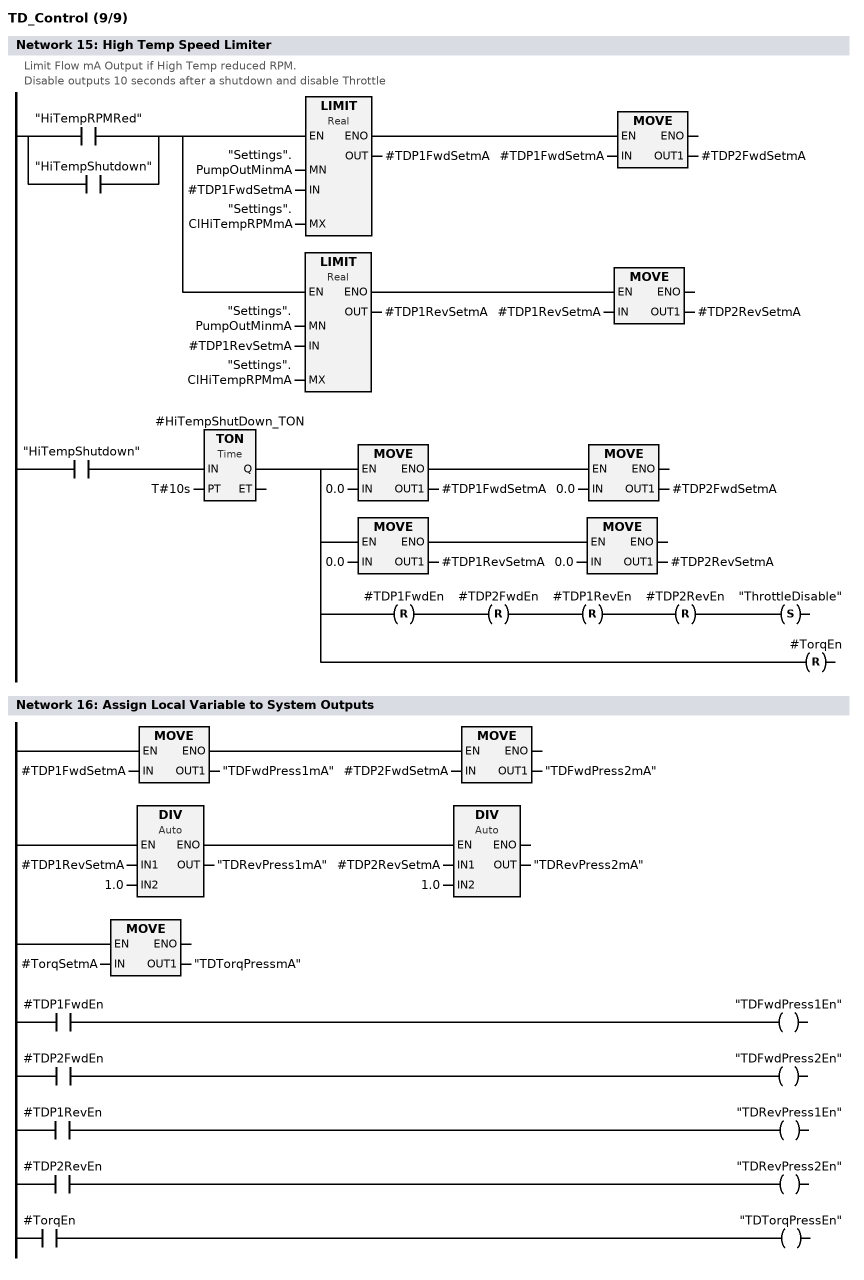
   RUNG wire#powerrail
      Contact( "HiTempRPMRed" )
      wire#w1
      { S7_Templates := "value_type := Real" } Limit(mn := "Settings".PumpOutMinmA, in := #TDP1FwdSetmA, mx := "Settings".ClHiTempRPMmA, out => #TDP1FwdSetmA)
      Move(in := #TDP1FwdSetmA, out1 => #TDP2FwdSetmA)
   END_RUNG
   RUNG wire#powerrail
      Contact( "HiTempShutdown" )
   END_RUNG wire#w1
   RUNG wire#w1
      { S7_Templates := "value_type := Real" } Limit(mn := "Settings".PumpOutMinmA, in := #TDP1RevSetmA, mx := "Settings".ClHiTempRPMmA, out => #TDP1RevSetmA)
      Move(in := #TDP1RevSetmA, out1 => #TDP2RevSetmA)
   END_RUNG
   RUNG wire#powerrail
      Contact( "HiTempShutdown" )
      { S7_Templates := "time_type := Time" } #HiTempShutDown_TON.TON(pt := T#10s, et =>)
      wire#w2
      Move(in := 0.0, out1 => #TDP1FwdSetmA)
      Move(in := 0.0, out1 => #TDP2FwdSetmA)
   END_RUNG
   RUNG wire#w2
      Move(in := 0.0, out1 => #TDP1RevSetmA)
      Move(in := 0.0, out1 => #TDP2RevSetmA)
   END_RUNG
   RUNG wire#w2
      R_Coil( #TDP1FwdEn )
      R_Coil( #TDP2FwdEn )
      R_Coil( #TDP1RevEn )
      R_Coil( #TDP2RevEn )
      S_Coil( "ThrottleDisable" )
   END_RUNG
   RUNG wire#w2
      R_Coil( #TorqEn )
   END_RUNG
   // the same network as SCL:
   IF "HiTempRPMRed" OR "HiTempShutdown" THEN
       #TDP1FwdSetmA := LIMIT(MN := "Settings".PumpOutMinmA, IN := #TDP1FwdSetmA, MX := "Settings".ClHiTempRPMmA);
       #TDP2FwdSetmA := #TDP1FwdSetmA;
       #TDP1RevSetmA := LIMIT(MN := "Settings".PumpOutMinmA, IN := #TDP1RevSetmA, MX := "Settings".ClHiTempRPMmA);
       #TDP2RevSetmA := #TDP1RevSetmA;
   END_IF;
   #HiTempShutDown_TON(IN := "HiTempShutdown", PT := T#10s);   // TON
   IF #HiTempShutDown_TON.Q THEN
       #TDP1FwdSetmA := 0.0;
       #TDP2FwdSetmA := 0.0;
       #TDP1RevSetmA := 0.0;
       #TDP2RevSetmA := 0.0;
       #TDP1FwdEn := FALSE;
       #TDP2FwdEn := FALSE;
       #TDP1RevEn := FALSE;
       #TDP2RevEn := FALSE;
       "ThrottleDisable" := TRUE;
       #TorqEn := FALSE;
   END_IF;
END_REGION

REGION Network 16: Assign Local Variable to System Outputs
   RUNG wire#powerrail
      Move(in := #TDP1FwdSetmA, out1 => "TDFwdPress1mA")
      Move(in := #TDP2FwdSetmA, out1 => "TDFwdPress2mA")
   END_RUNG
   RUNG wire#powerrail
      Div(in1 := #TDP1RevSetmA, in2 := 1.0, out => "TDRevPress1mA")
      Div(in1 := #TDP2RevSetmA, in2 := 1.0, out => "TDRevPress2mA")
   END_RUNG
   RUNG wire#powerrail
      Move(in := #TorqSetmA, out1 => "TDTorqPressmA")
   END_RUNG
   RUNG wire#powerrail
      Contact( #TDP1FwdEn )
      Coil( "TDFwdPress1En" )
   END_RUNG
   RUNG wire#powerrail
      Contact( #TDP2FwdEn )
      Coil( "TDFwdPress2En" )
   END_RUNG
   RUNG wire#powerrail
      Contact( #TDP1RevEn )
      Coil( "TDRevPress1En" )
   END_RUNG
   RUNG wire#powerrail
      Contact( #TDP2RevEn )
      Coil( "TDRevPress2En" )
   END_RUNG
   RUNG wire#powerrail
      Contact( #TorqEn )
      Coil( "TDTorqPressEn" )
   END_RUNG
   // the same network as SCL:
   "TDFwdPress1mA" := #TDP1FwdSetmA;
   "TDFwdPress2mA" := #TDP2FwdSetmA;
   "TDRevPress1mA" := #TDP1RevSetmA / 1.0;
   "TDRevPress2mA" := #TDP2RevSetmA / 1.0;
   "TDTorqPressmA" := #TorqSetmA;
   "TDFwdPress1En" := #TDP1FwdEn;
   "TDFwdPress2En" := #TDP2FwdEn;
   "TDRevPress1En" := #TDP1RevEn;
   "TDRevPress2En" := #TDP2RevEn;
   "TDTorqPressEn" := #TorqEn;
END_REGION
END_FUNCTION_BLOCK
